TYPE ST_Recipe :
STRUCT
	RequiredChargedV : REAL := 10;
END_STRUCT
END_TYPE

(* stored: Version 1.1.0.1, ProductVersion 3.1.4024.11
   DUT ST_Recipe: Id {2065798b-e446-4a94-ba0f-3197caff863b} *)
